TYPE ST_PNInput_InputGridControl :
STRUCT
	w_Control				:	WORD;
	ui_FeedInCurrentLimit	:	UINT;
	ui_SupplyCurrentLimit	:	UINT;
	ui_CurrentLimitRetries	:	UINT;
	ui_ContactorControl		:	uint;
END_STRUCT
END_TYPE

(* stored: Version 1.1.0.1, ProductVersion 3.1.4026.18
   DUT ST_PNInput_InputGridControl: Id {27ace1a5-3d45-4e45-9fd2-e49196a4f393} *)
